// TIA Portal V15 export
// export: Created 2018-05-29T12:25:38.1552518Z, ExportSetting WithDefaults, DisplayName Totally Integrated Automation Portal, DisplayVersion V15, DisplayName STEP 7 Professional, DisplayVersion V15, DisplayName WinCC Professional, DisplayVersion V15, DisplayName TIA Portal Openness, DisplayVersion V15
FUNCTION "em_write" : Void   // FC1, STL
{ S7_Optimized_Access := 'FALSE' }
VERSION : 0.1
// stored: AutoNumber true, UDAEnableTagReadback false
   VAR_INPUT
      EM_ID : Int;
      UDT_LOCATION : Pointer;
      UDT_OFFSET : Int;
      Length : Int;
      Request : Int;
      Owner : Int;
   END_VAR
   VAR_OUTPUT
      EM_addressing_error : Bool;
   END_VAR
   VAR_TEMP
      em_address : Int;
      em_index_length : Int;
      em_db : Int;
      em_udt : Int;
      phase_db : Int;
      phase_udt : Int;
      source_pointer : Any;
      dest_pointer : Any;
      adjusted_length : Int;
      blkmov_retval : Int;
   END_VAR
BEGIN

NETWORK
TITLE = 

// Skip the entire FC if Request = 0

      L     #Request;
      L     0;
      ==I;
      JCN   ENDS;

// Reduce the length to one Integer if the EM has not been acquired yet
      L     #Owner;
      L     #Request;
      <>I;
      JCN   REDU;

      L     2;
      T     #adjusted_length;

REDU: NOP   0;


// Calculate the amount of EMs in the EM_Index
      OPN   "db25";
      L     DBLG;
      L     4;
      /I;
      T     #em_index_length;


// protect against an address outside db25
      L     #EM_ID;
      L     #em_index_length;
      >I;
      =     #EM_addressing_error;
      JC    ENDS;


// calculate the address of the EM in DB25
      L     #EM_ID;
      L     4;
      *I;
      T     #em_address;

// prepare the pointer for the location in EM Index DB
// todo: probably don't need to load the 0-pointer
      L     P#DBX0.0;
      L     #em_address;
      SLD   3;
      +D;
      LAR1;

// read the DB number
      L     DBW [AR1, P#0.0];
      T     #em_db;

// read the UDT location
      L     DBW [AR1, P#2.0];
      T     #em_udt;

// read the start of the UDT in the phase
      L     P##UDT_LOCATION;
      LAR1;
      L     DBD [AR1, P#2.0];
      L     DW#16#7FFF8;
      AD;
      SRD   3;
      T     #phase_udt;

// read the phase DB
      L     DBW [AR1, P#0.0];
      T     #phase_db;

// prepare the receiving address
      LAR1  P##dest_pointer;
      L     W#16#1002;  //Syntax ID (10h for S7, 2h bytes)
      T     DBW [AR1, P#0.0];
      L     #adjusted_length;  //Length in bytes
      T     DBW [AR1, P#2.0];
      L     #em_db;  //DB-nummer EM
      T     DBW [AR1, P#4.0];
      L     #em_udt;  //Start address in DB EM
      L     #UDT_OFFSET;
      +I;
      SLD   3;
      L     DW#16#84000000;
      OD;
      T     DBD [AR1, P#6.0];

// prepare the sending address
      LAR1  P##source_pointer;
      L     W#16#1002;  //Syntax ID (10h for S7, 2h bytes)
      T     DBW [AR1, P#0.0];
      L     #adjusted_length;  //Length in bytes
      T     DBW [AR1, P#2.0];
      L     #phase_db;  //DB-nummer SEQ
      T     DBW [AR1, P#4.0];
      L     #phase_udt;  //Start address in DB SEQ
      L     #UDT_OFFSET;
      +I;
      SLD   3;
      L     DW#16#84000000;
      OD;
      T     DBD [AR1, P#6.0];

// copy the data
      CALL  BLKMOV
      ( SRCBLK  := #source_pointer,
        RET_VAL := #blkmov_retval,
        DSTBLK  := #dest_pointer
      );




ENDS: NOP   0;


END_FUNCTION
